(* IEC 61131-3 sources: teller/JD_Teller_LC2_V11/Class/Signal_Splitter, 1 file *)

(* ---- Signal_Splitter.st ---- *)
(*!
<Class
	Name               = "Signal_Splitter"
	Revision           = "0.0"
	RealtimeTask       = "false"
	CyclicTask         = "false"
	BackgroundTask     = "false"
	Sigmatek           = "false"
	OSInterface        = "false"
	HighPriority       = "false"
	Automatic          = "false"
	UpdateMode         = "Prescan"
	SharedCommandTable = "true"
	Objectsize         = "(540,120)">
	<Channels>
		<Server Name="ClassSvr" Visualized="false" Initialize="false" WriteProtected="true" Retentive="false"/>
		<Server Name="WriteValue" Visualized="true" Initialize="false" WriteProtected="false" Retentive="false"/>
		<Client Name="c_WriteValue01" Required="false" Internal="false"/>
		<Client Name="c_WriteValue02" Required="false" Internal="false"/>
		<Client Name="c_WriteValue03" Required="false" Internal="false"/>
		<Client Name="c_WriteValue04" Required="false" Internal="false"/>
		<Client Name="c_WriteValue05" Required="false" Internal="false"/>
		<Client Name="c_WriteValue06" Required="false" Internal="false"/>
		<Client Name="c_WriteValue07" Required="false" Internal="false"/>
		<Client Name="c_WriteValue08" Required="false" Internal="false"/>
		<Client Name="c_WriteValue09" Required="false" Internal="false"/>
		<Client Name="c_WriteValue10" Required="false" Internal="false"/>
		<Client Name="c_WriteValue11" Required="false" Internal="false"/>
		<Client Name="c_WriteValue12" Required="false" Internal="false"/>
	</Channels>
</Class>
*)
Signal_Splitter : CLASS
  //Servers:
	ClassSvr 	: SvrChCmd_DINT;
	WriteValue 	: SvrCh_DINT;
  //Clients:
	c_WriteValue01 	: CltCh_DINT;
	c_WriteValue02 	: CltCh_DINT;
	c_WriteValue03 	: CltCh_DINT;
	c_WriteValue04 	: CltCh_DINT;
	c_WriteValue05 	: CltCh_DINT;
	c_WriteValue06 	: CltCh_DINT;
	c_WriteValue07 	: CltCh_DINT;
	c_WriteValue08 	: CltCh_DINT;
	c_WriteValue09 	: CltCh_DINT;
	c_WriteValue10 	: CltCh_DINT;
	c_WriteValue11 	: CltCh_DINT;
	c_WriteValue12 	: CltCh_DINT;
  //Variables:
  //Functions:

	FUNCTION VIRTUAL GLOBAL WriteValue::Write
		VAR_INPUT
			input (EAX) 	: DINT;
		END_VAR
		VAR_OUTPUT
			result (EAX) 	: DINT;
		END_VAR;
  //Tables:
	FUNCTION @STD
		VAR_OUTPUT
			ret_code	: CONFSTATES;
		END_VAR;
	FUNCTION GLOBAL TAB @CT_;
END_CLASS;

FUNCTION VIRTUAL GLOBAL Signal_Splitter::WriteValue::Write
	VAR_INPUT
		input (EAX) 	: DINT;
	END_VAR
	VAR_OUTPUT
		result (EAX) 	: DINT;
	END_VAR

	WriteValue := input;

  c_WriteValue01.Write (WriteValue);
  c_WriteValue02.Write (WriteValue);
  c_WriteValue03.Write (WriteValue);
  c_WriteValue04.Write (WriteValue);
  c_WriteValue05.Write (WriteValue);
  c_WriteValue06.Write (WriteValue);
  c_WriteValue07.Write (WriteValue);
  c_WriteValue08.Write (WriteValue);
  c_WriteValue09.Write (WriteValue);
  c_WriteValue10.Write (WriteValue);
  c_WriteValue11.Write (WriteValue);
  c_WriteValue12.Write (WriteValue);

 	result := WriteValue;

END_FUNCTION
